// Mitsubishi GX Works2 project: LRI - PLC - AULA 10   PLC: Q03UDV

// task Task_01 (event TRUE, interval 0, priority 31): POU_01

PROGRAM POU_01
VAR
  diResult : DINT;
  diResultDiv : ARRAY [0..1] OF INT;
END_VAR
(* structured ladder/FBD written out as ST: instructions are called as NAME(EN, inputs, outputs); _pN, _eN, _tN stand for wires *)
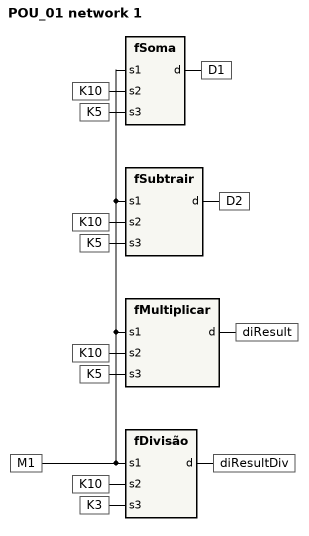
(* network 1 *)
D1 := fSoma(M1, K10, K5);
D2 := fSubtrair(M1, K10, K5);
diResult := fMultiplicar(M1, K10, K5);
diResultDiv := fDivisão(M1, K10, K3);
END_PROGRAM

FUNCTION fSoma
VAR_INPUT
  i_xHabilitar : BOOL;
  i_iVariavelUm : INT;
  i_iVariavelDois : INT;
END_VAR
(* structured ladder/FBD written out as ST: instructions are called as NAME(EN, inputs, outputs); _pN, _eN, _tN stand for wires *)
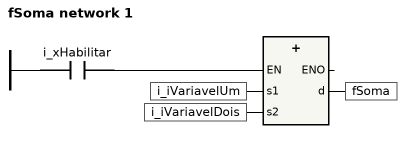
(* network 1 *)
+(i_xHabilitar, i_iVariavelUm, i_iVariavelDois, fSoma);
END_FUNCTION

FUNCTION fSubtrair
VAR_INPUT
  i_xHabilitarSubtrair : BOOL;
  i_iVariavelUmSubtrair : INT;
  i_iVariavelDoisSubtrair : INT;
END_VAR
(* structured ladder/FBD written out as ST: instructions are called as NAME(EN, inputs, outputs); _pN, _eN, _tN stand for wires *)
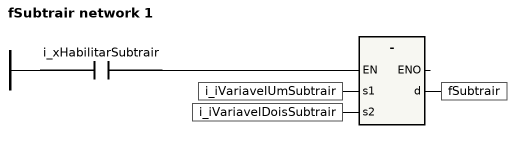
(* network 1 *)
-(i_xHabilitarSubtrair, i_iVariavelUmSubtrair, i_iVariavelDoisSubtrair, fSubtrair);
END_FUNCTION

FUNCTION fMultiplicar
VAR_INPUT
  i_xHabilitarMultiplicar : BOOL;
  i_iVariavelUmMultiplicar : INT;
  i_iVariavelDoisMultiplicar : INT;
END_VAR
(* structured ladder/FBD written out as ST: instructions are called as NAME(EN, inputs, outputs); _pN, _eN, _tN stand for wires *)
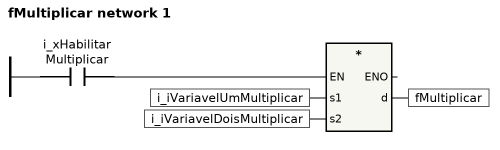
(* network 1 *)
*(i_xHabilitarMultiplicar, i_iVariavelUmMultiplicar, i_iVariavelDoisMultiplicar, fMultiplicar);
END_FUNCTION

FUNCTION fDivisão
VAR_INPUT
  i_xHabilitarDividir : BOOL;
  i_iVariavelUmDividir : INT;
  i_iVariavelDoisDividir : INT;
END_VAR
(* structured ladder/FBD written out as ST: instructions are called as NAME(EN, inputs, outputs); _pN, _eN, _tN stand for wires *)
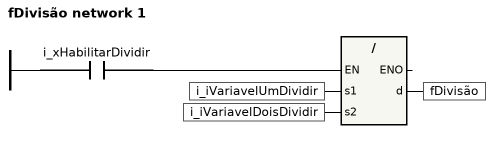
(* network 1 *)
/(i_xHabilitarDividir, i_iVariavelUmDividir, i_iVariavelDoisDividir, fDivisão);
END_FUNCTION

FUNCTION_BLOCK fbBlink
END_FUNCTION_BLOCK
